ABB RAPID module: HSLU_Workobject.modx

MODULE HSLU_Workobject

    !***********************************************************************************
    !
    ! Digital Construction
    ! Hochschule Luzern - Technik & Architektur
    ! Technikumstrasse 21
    ! CH-6048 Horw
    !
    !***********************************************************************************
    !
    ! PROJECT     :  Swissbau
    !
    ! FUNCTION    :  Workobject
    !
    ! AUTHOR      :  Juri Jerg
    !
    ! EMAIL       :  juri.jerg@hslu.ch
    !
    ! HISTORY     :  2025.12.28
    !
    ! Copyright   :  HSLU (2025)
    !
    !***********************************************************************************

    !************************************************
    ! Declaration :     wobjdata
    !************************************************
    !
    TASK PERS wobjdata ob_HSLU_Pick := [FALSE,TRUE,"",[[1140.146,313.9341,-37.721858],[0.001277417,0.001486036,-0.007628683,-0.999969]],[[0,0,0],[1,0,0,0]]];
    !TASK PERS wobjdata ob_HSLU_Cut := [FALSE,TRUE,"",[[418.7775,-1110.276,-31.90539],[0.7049414,0.001132027,-0.002334736,-0.7092608]],[[0,0,0],[1,0,0,0]]];
    !TASK PERS wobjdata ob_HSLU_Cut := [FALSE,TRUE,"",[[515.455,-1126.729,-1.878],[0.7049414,0.001132027,-0.002334736,-0.7092608]],[[0,0,0],[1,0,0,0]]];
    !TASK PERS wobjdata ob_HSLU_Cut := [FALSE,TRUE,"",[[565.30654095,-1126.982741334,28.366990995],[0.704941403,0.001132027,-0.002334736,-0.709260803]],[[0,0,0],[1,0,0,0]]];
    !TASK PERS wobjdata ob_HSLU_Cut := [FALSE,TRUE,"",[[615.305007167,-1127.287958109,28.612385938],[0.704941403,0.001132027,-0.002334736,-0.709260803]],[[0,0,0],[1,0,0,0]]];
    TASK PERS wobjdata ob_HSLU_Cut := [FALSE,TRUE,"",[[328.0311,-1088.269,-37.87487],[0.7055837,0.0007998496,-0.002891258,-0.7086203]],[[13.368,192.018,72.161],[1,0,0,0]]];
    TASK PERS wobjdata ob_HSLU_Place := [FALSE,TRUE,"",[[460,0,1],[0.707106781,0,0,0.707106781]],[[0,0,0],[1,0,0,0]]];
    TASK PERS wobjdata ob_HSLU_Glue := [FALSE,TRUE,"",[[460,-1000,1500],[0,0.707106781,0.707106781,0]],[[0,0,0],[1,0,0,0]]];
    TASK PERS wobjdata ob_HSLU_Lable := [FALSE,TRUE,"",[[460,-1000,1000],[0,0.707106781,0.707106781,0]],[[0,0,0],[1,0,0,0]]];
ENDMODULE
